{attribute 'qualified_only'}
VAR_GLOBAL
	b_yellow_button		AT %I* :BOOL;
	b_blue_button		AT %I* :BOOL;
	b_green_lamp		AT %Q* :BOOL;
	b_red_lamp			AT %Q* :BOOL;
END_VAR

(* stored: Version 1.1.0.1, ProductVersion 3.1.4022.12
   GVL GVL_IO: Id {a5726f5c-cc2c-4806-ac29-43fb6f35813b} *)
